ABB RobotStudio station: EstaciónDeSoldadura_20200720-232522.rsstn

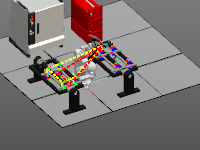
Station EstaciónDeSoldadura (saved by RobotStudio 7.0.8746.631)
Controller IRB_140_6kg_0.81m
  mechanical unit ROB_1: IRB140_6_81_C_03, 6 joints, base frame (0, 0, 0) mm
Layout (positions relative to the parent item):
  - IRB140_6_81_C_03 [mechanism, from Robots\IRB140_6_81_C_G_03.rslib] at (0, 0, 0) mm; joint values [0, 0, -0.7854, 0, 0, 0] (rad or m)
  - AW_Gun_PSF_25 [mechanism, from Tools\AW_Gun_PSF_25.rslib] at (384.66, 0, 1026.66) mm, rotated rx 0 ry 45 rz 0 deg
  - IRC5_Singel-Cabinet [part, from Equipment\IRC5_Singel-Cabinet.rslib] at (-1350, 0, 100) mm, rotated rx 90 ry 0 rz 90 deg
  - Fronius_TPS4000_rev0 [part, from Equipment\Fronius_TPS4000.rslib] at (-1350, 900, 0) mm, rotated rx 0 ry 0 rz -90 deg
  - FlexPendant [part, from Equipment\FlexPendant.rslib] at (-1350, 0, 1100) mm, rotated rx 0 ry 0 rz 90 deg
  - Mesa [mechanism] at (-540, -540, 0) mm; joint values [0] (rad or m)
      links: L1, L2, L3
  - Mesa_2 [mechanism] at (-540, 540, 0) mm; joint values [0] (rad or m)
      links: L1, L2, L3
Attachment: AW_Gun_PSF_25 is attached to IRB140_6_81_C_03 / Link6
Attachment: Workobject_Mesa1 is attached to Mesa / L2
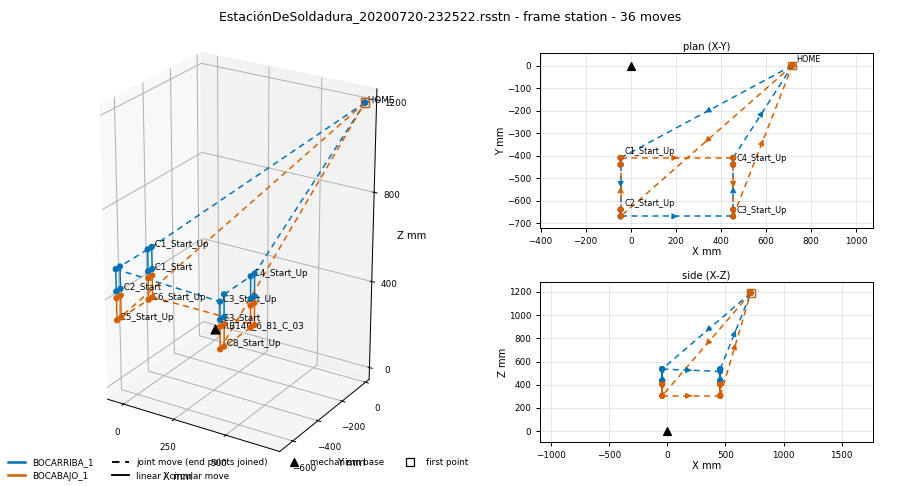
[picture p0: tool path of EstaciónDeSoldadura_20200720-232522.rsstn in frame station, 36 of 36 moves have a stored position in this frame; points joined in program order, loops and branches not executed]
Targets, tools, work objects and paths stored in the station, written as RAPID:
! task T_ROB1
MODULE CalibData
  PERS tooldata AW_Gun:=[TRUE,[[119.5,0,352],[0.890213743,0,0.455543074,0]],[1,[0,0,100],[1,0,0,0],0,0,0]];
  PERS wobjdata Workobject_Mesa1:=[FALSE,TRUE,"",[[-590,-540,370],[0.707106781,0.707106781,0,0]],[[0,0,0],[1,0,0,0]]];
ENDMODULE

! task T_ROB1
MODULE Module1
  CONST robtarget C1_Start:=[[545,65,-130],[0.5,0.5,0.5,-0.5],[-2,0,-1,0],[9E+09,9E+09,9E+09,9E+09,9E+09,9E+09]];
  CONST robtarget C1_Final:=[[545,65,-100],[0.5,0.5,0.5,-0.5],[-2,0,-1,0],[9E+09,9E+09,9E+09,9E+09,9E+09,9E+09]];
  CONST robtarget C2_Start:=[[545,65,100],[0.5,0.5,0.5,-0.5],[-2,0,-1,0],[9E+09,9E+09,9E+09,9E+09,9E+09,9E+09]];
  CONST robtarget C2_Final:=[[545,65,130],[0.5,0.5,0.5,-0.5],[-2,0,-1,0],[9E+09,9E+09,9E+09,9E+09,9E+09,9E+09]];
  CONST robtarget C3_Start:=[[1045,65,130],[0.5,0.5,0.5,-0.5],[-1,-1,0,0],[9E+09,9E+09,9E+09,9E+09,9E+09,9E+09]];
  CONST robtarget C3_Final:=[[1045,65,100],[0.5,0.5,0.5,-0.5],[-1,-1,0,0],[9E+09,9E+09,9E+09,9E+09,9E+09,9E+09]];
  CONST robtarget C4_Start:=[[1045,65,-100],[0.5,0.5,0.5,-0.5],[-1,-1,0,0],[9E+09,9E+09,9E+09,9E+09,9E+09,9E+09]];
  CONST robtarget C4_Final:=[[1045,65,-130],[0.5,0.5,0.5,-0.5],[-1,-1,0,0],[9E+09,9E+09,9E+09,9E+09,9E+09,9E+09]];
  CONST robtarget C1_Final_Up:=[[545,165,-100],[0.5,0.5,0.5,-0.5],[-2,0,-1,0],[9E+09,9E+09,9E+09,9E+09,9E+09,9E+09]];
  CONST robtarget C1_Start_Up:=[[545.000020572,165.000017529,-129.999987486],[0.500000003,0.499999966,0.499999998,-0.500000033],[-2,0,-1,0],[9E+09,9E+09,9E+09,9E+09,9E+09,9E+09]];
  CONST robtarget C2_Final_Up:=[[545,165,130],[0.5,0.5,0.5,-0.5],[-2,0,-1,0],[9E+09,9E+09,9E+09,9E+09,9E+09,9E+09]];
  CONST robtarget C2_Start_Up:=[[545,165,100],[0.5,0.5,0.5,-0.5],[-2,0,-1,0],[9E+09,9E+09,9E+09,9E+09,9E+09,9E+09]];
  CONST robtarget C3_Final_Up:=[[1045,165,100],[0.5,0.5,0.5,-0.5],[-1,-1,0,0],[9E+09,9E+09,9E+09,9E+09,9E+09,9E+09]];
  CONST robtarget C3_Start_Up:=[[1045.000011824,144.999988637,130.000030031],[0.500000021,0.499999969,0.499999973,-0.500000036],[-2,0,-1,0],[9E+09,9E+09,9E+09,9E+09,9E+09,9E+09]];
  CONST robtarget C4_Final_Up:=[[1045,165,-130],[0.5,0.5,0.5,-0.5],[-1,-1,0,0],[9E+09,9E+09,9E+09,9E+09,9E+09,9E+09]];
  CONST robtarget C4_Start_Up:=[[1045,165,-100],[0.5,0.5,0.5,-0.5],[-1,-1,0,0],[9E+09,9E+09,9E+09,9E+09,9E+09,9E+09]];
  CONST robtarget C5_Start:=[[545,35,130],[0.5,-0.5,-0.5,-0.5],[-2,0,-1,0],[9E+09,9E+09,9E+09,9E+09,9E+09,9E+09]];
  CONST robtarget C5_Final:=[[545,35,100],[0.5,-0.5,-0.5,-0.5],[-2,0,-1,0],[9E+09,9E+09,9E+09,9E+09,9E+09,9E+09]];
  CONST robtarget C6_Start:=[[545,35,-100],[0.5,-0.5,-0.5,-0.5],[-2,0,-1,0],[9E+09,9E+09,9E+09,9E+09,9E+09,9E+09]];
  CONST robtarget C6_Final:=[[545,35,-130],[0.5,-0.5,-0.5,-0.5],[-2,0,-1,0],[9E+09,9E+09,9E+09,9E+09,9E+09,9E+09]];
  CONST robtarget C7_Start:=[[1045,35,-130],[0.5,-0.5,-0.5,-0.5],[-1,-1,0,0],[9E+09,9E+09,9E+09,9E+09,9E+09,9E+09]];
  CONST robtarget C7_Final:=[[1045,35,-100],[0.5,-0.5,-0.5,-0.5],[-1,-1,0,0],[9E+09,9E+09,9E+09,9E+09,9E+09,9E+09]];
  CONST robtarget C8_Start:=[[1045,35,100],[0.5,-0.5,-0.5,-0.5],[-1,-1,0,0],[9E+09,9E+09,9E+09,9E+09,9E+09,9E+09]];
  CONST robtarget C8_Final:=[[1045,35,130],[0.5,-0.5,-0.5,-0.5],[-1,-1,0,0],[9E+09,9E+09,9E+09,9E+09,9E+09,9E+09]];
  CONST robtarget C5_Final_Up:=[[545,-65,100],[0.5,-0.5,-0.5,-0.5],[-2,0,-1,0],[9E+09,9E+09,9E+09,9E+09,9E+09,9E+09]];
  CONST robtarget C5_Start_Up:=[[545,-65,130],[0.5,-0.5,-0.5,-0.5],[-2,0,-1,0],[9E+09,9E+09,9E+09,9E+09,9E+09,9E+09]];
  CONST robtarget C6_Final_Up:=[[545,-65,-130],[0.5,-0.5,-0.5,-0.5],[-2,0,-1,0],[9E+09,9E+09,9E+09,9E+09,9E+09,9E+09]];
  CONST robtarget C6_Start_Up:=[[545,-65,-100],[0.5,-0.5,-0.5,-0.5],[-2,0,-1,0],[9E+09,9E+09,9E+09,9E+09,9E+09,9E+09]];
  CONST robtarget C7_Final_Up:=[[1045,-65,-100],[0.5,-0.5,-0.5,-0.5],[-1,-1,0,0],[9E+09,9E+09,9E+09,9E+09,9E+09,9E+09]];
  CONST robtarget C7_Start_Up:=[[1045,-65,-130],[0.5,-0.5,-0.5,-0.5],[-1,-1,0,0],[9E+09,9E+09,9E+09,9E+09,9E+09,9E+09]];
  CONST robtarget C8_Final_Up:=[[1045,-65,130],[0.5,-0.5,-0.5,-0.5],[0,0,0,0],[9E+09,9E+09,9E+09,9E+09,9E+09,9E+09]];
  CONST robtarget C8_Start_Up:=[[1045,-65,100],[0.5,-0.5,-0.5,-0.5],[-1,-1,0,0],[9E+09,9E+09,9E+09,9E+09,9E+09,9E+09]];
  CONST robtarget HOME:=[[718.063364957,0,1191.064844254],[0.648121469,0,0.761536973,0],[0,0,0,0],[9E+09,9E+09,9E+09,9E+09,9E+09,9E+09]];
  CONST robtarget HOME_2:=[[718.063364957,0,1191.064844254],[0.648121469,0,0.761536973,0],[0,0,0,0],[9E+09,9E+09,9E+09,9E+09,9E+09,9E+09]];
  CONST robtarget C12_Start:=[[-45,410,435],[0,-0.707106781,0.707106781,0],[0,0,0,0],[9E+09,9E+09,9E+09,9E+09,9E+09,9E+09]];
  CONST robtarget C12_Final:=[[-45,440,435],[0,-0.707106781,0.707106781,0],[0,0,0,0],[9E+09,9E+09,9E+09,9E+09,9E+09,9E+09]];
  CONST robtarget C22_Start:=[[-45,640,435],[0,-0.707106781,0.707106781,0],[0,0,0,0],[9E+09,9E+09,9E+09,9E+09,9E+09,9E+09]];
  CONST robtarget C22_Final:=[[-45,670,435],[0,-0.707106781,0.707106781,0],[0,0,0,0],[9E+09,9E+09,9E+09,9E+09,9E+09,9E+09]];
  CONST robtarget C32_Start:=[[455,670,435],[0,-0.707106781,0.707106781,0],[0,0,0,0],[9E+09,9E+09,9E+09,9E+09,9E+09,9E+09]];
  CONST robtarget C32_Final:=[[455,640,435],[0,-0.707106781,0.707106781,0],[0,0,0,0],[9E+09,9E+09,9E+09,9E+09,9E+09,9E+09]];
  CONST robtarget C42_Start:=[[455,440,435],[0,-0.707106781,0.707106781,0],[0,0,0,0],[9E+09,9E+09,9E+09,9E+09,9E+09,9E+09]];
  CONST robtarget C42_Final:=[[455,410,435],[0,-0.707106781,0.707106781,0],[0,0,0,0],[9E+09,9E+09,9E+09,9E+09,9E+09,9E+09]];
  CONST robtarget C12_Final_Up:=[[-45,440,535],[0,-0.707106781,0.707106781,0],[0,0,0,0],[9E+09,9E+09,9E+09,9E+09,9E+09,9E+09]];
  CONST robtarget C12_Start_Up:=[[-45,410,535],[0,-0.707106781,0.707106781,0],[0,0,0,0],[9E+09,9E+09,9E+09,9E+09,9E+09,9E+09]];
  CONST robtarget C22_Final_Up:=[[-45,670,535],[0,-0.707106781,0.707106781,0],[0,0,0,0],[9E+09,9E+09,9E+09,9E+09,9E+09,9E+09]];
  CONST robtarget C22_Start_Up:=[[-45,640,535],[0,-0.707106781,0.707106781,0],[0,0,0,0],[9E+09,9E+09,9E+09,9E+09,9E+09,9E+09]];
  CONST robtarget C32_Final_Up:=[[455,640,535],[0,-0.707106781,0.707106781,0],[0,0,0,0],[9E+09,9E+09,9E+09,9E+09,9E+09,9E+09]];
  CONST robtarget C32_Start_Up:=[[455,670,515],[0,-0.707106781,0.707106781,0],[0,0,0,0],[9E+09,9E+09,9E+09,9E+09,9E+09,9E+09]];
  CONST robtarget C42_Final_Up:=[[455,410,535],[0,-0.707106781,0.707106781,0],[0,0,0,0],[9E+09,9E+09,9E+09,9E+09,9E+09,9E+09]];
  CONST robtarget C42_Start_Up:=[[455,440,535],[0,-0.707106781,0.707106781,0],[0,0,0,0],[9E+09,9E+09,9E+09,9E+09,9E+09,9E+09]];
  CONST robtarget HOME_3:=[[718.063364957,0,1191.064844254],[0.648121469,0,0.761536973,0],[0,0,0,0],[9E+09,9E+09,9E+09,9E+09,9E+09,9E+09]];
  CONST robtarget HOME_3_3:=[[718.063364957,0,1191.064844254],[0.648121469,0,0.761536973,0],[0,0,0,0],[9E+09,9E+09,9E+09,9E+09,9E+09,9E+09]];
  CONST robtarget HOME_4:=[[718.063364957,0,1191.064844254],[0.648121469,0,0.761536973,0],[0,0,0,0],[9E+09,9E+09,9E+09,9E+09,9E+09,9E+09]];
  PROC main()
  ENDPROC
  PROC BOCARRIBA_1()
    MoveJ HOME,v3000,z100,AW_Gun\WObj:=wobj0;
    MoveJ C1_Start_Up,v1000,z100,AW_Gun\WObj:=Workobject_Mesa1;
    MoveL C1_Start,v200,z0,AW_Gun\WObj:=Workobject_Mesa1;
    MoveL C1_Final,v10,z0,AW_Gun\WObj:=Workobject_Mesa1;
    MoveL C1_Final_Up,v200,z0,AW_Gun\WObj:=Workobject_Mesa1;
    MoveJ C2_Start_Up,v1000,z100,AW_Gun\WObj:=Workobject_Mesa1;
    MoveL C2_Start,v200,z0,AW_Gun\WObj:=Workobject_Mesa1;
    MoveL C2_Final,v10,z0,AW_Gun\WObj:=Workobject_Mesa1;
    MoveL C2_Final_Up,v200,z0,AW_Gun\WObj:=Workobject_Mesa1;
    MoveJ C3_Start_Up,v1000,z100,AW_Gun\WObj:=Workobject_Mesa1;
    MoveL C3_Start,v200,z0,AW_Gun\WObj:=Workobject_Mesa1;
    MoveL C3_Final,v10,z0,AW_Gun\WObj:=Workobject_Mesa1;
    MoveL C3_Final_Up,v200,z0,AW_Gun\WObj:=Workobject_Mesa1;
    MoveJ C4_Start_Up,v1000,z100,AW_Gun\WObj:=Workobject_Mesa1;
    MoveL C4_Start,v200,z0,AW_Gun\WObj:=Workobject_Mesa1;
    MoveL C4_Final,v10,z0,AW_Gun\WObj:=Workobject_Mesa1;
    MoveL C4_Final_Up,v200,z0,AW_Gun\WObj:=Workobject_Mesa1;
    MoveJ HOME_4,v3000,z100,AW_Gun\WObj:=wobj0;
  ENDPROC
  PROC BOCABAJO_1()
    MoveJ HOME_2,v3000,z100,AW_Gun\WObj:=wobj0;
    MoveJ C5_Start_Up,v1000,z100,AW_Gun\WObj:=Workobject_Mesa1;
    MoveL C5_Start,v200,z0,AW_Gun\WObj:=Workobject_Mesa1;
    MoveL C5_Final,v10,z0,AW_Gun\WObj:=Workobject_Mesa1;
    MoveL C5_Final_Up,v200,z0,AW_Gun\WObj:=Workobject_Mesa1;
    MoveJ C6_Start_Up,v1000,z100,AW_Gun\WObj:=Workobject_Mesa1;
    MoveL C6_Start,v200,z0,AW_Gun\WObj:=Workobject_Mesa1;
    MoveL C6_Final,v10,z0,AW_Gun\WObj:=Workobject_Mesa1;
    MoveL C6_Final_Up,v200,z0,AW_Gun\WObj:=Workobject_Mesa1;
    MoveJ C7_Start_Up,v1000,z100,AW_Gun\WObj:=Workobject_Mesa1;
    MoveL C7_Start,v200,z0,AW_Gun\WObj:=Workobject_Mesa1;
    MoveL C7_Final,v10,z0,AW_Gun\WObj:=Workobject_Mesa1;
    MoveL C7_Final_Up,v200,z0,AW_Gun\WObj:=Workobject_Mesa1;
    MoveJ C8_Start_Up,v1000,z100,AW_Gun\WObj:=Workobject_Mesa1;
    MoveL C8_Start,v200,z0,AW_Gun\WObj:=Workobject_Mesa1;
    MoveL C8_Final,v10,z0,AW_Gun\WObj:=Workobject_Mesa1;
    MoveL C8_Final_Up,v200,z0,AW_Gun\WObj:=Workobject_Mesa1;
    MoveJ HOME_2,v3000,z100,AW_Gun\WObj:=wobj0;
  ENDPROC
ENDMODULE

